// TIA Portal V18 export
DATA_BLOCK "deletemot_speed_wdir_slowly_accelerated_DB"   // DB39
VERSION : 0.1
// stored: AutoNumber true, DBAccessibleFromOPCUA true, InstanceOfName mot_speed_wdir_slowly_accelerated, InstanceOfType FB
"mot_speed_wdir_slowly_accelerated"
   // VAR_INPUT
   //    ALLOWED : Bool;
   //    set_speed__wdir : Real;
   //    v_absMax : Real;
   //    t_acc : Real;
   //    STOP_NOW : Bool;
   // END_VAR
   // VAR_OUTPUT
   //    speed_accelerated_slowly_wdir : Real;
   // END_VAR
   // VAR
   //    speed_is_zero : Bool;
   //    speed_is_zero_was : Bool;
   //    speed_is_zero_CLK : Bool;
   // END_VAR
BEGIN
END_DATA_BLOCK
